(* Logix 5000 project; controller R1USB70001_CWRU_Scenario_Gen_20111116 vendor 1 type 14 code 54 rev 19.11; software revision 19.01 *)

TASK MainTask (continuous, watchdog 500 ms) : MainProgram

MODULES
   Local : vendor 1 type 14 code 54 (ICP 2, rev 19.11)
      CNB_Scenario_Generator : vendor 1 type 12 code 21 (ICP 0, rev 20.13)
         ACNR_SP_SG_N3 : vendor 1 type 12 code 111 (ControlNet 3, rev 1.83, Output RPI 8 ms)
            OB8_SP_SG_S3 : 1734-OE2V (PointIO 3, rev 3.5, Output RPI 8 ms)
            OB8_SP_SG_S2 : 1734-OB8 (PointIO 2, rev 3.22)
            OB8_SP_SG_S1 : 1734-OB8 (PointIO 1, rev 3.22)
         ACNR_RP_SG_N4 : vendor 1 type 12 code 111 (ControlNet 4, rev 1.83, Output RPI 8 ms)
            OB8_RP_SG_S1 : 1734-OB8 (PointIO 1, rev 3.22)
            OB8_RP_SG_S2 : 1734-OB8 (PointIO 2, rev 3.22)
            OB8_RP_SG_S3 : 1734-OB8 (PointIO 3, rev 3.22)
            OB8_RP_SG_S5 : 1734-OB8 (PointIO 5, rev 3.22)
            OB8_RP_SG_S6 : 1734-OB8 (PointIO 6, rev 3.22)
            OB8_RP_SG_S4 : 1734-OB8 (PointIO 4, rev 3.22)
         ACNR_GP_SG_N2 : vendor 1 type 12 code 111 (ControlNet 2, rev 1.83, Output RPI 8 ms)
            OB8_GP_SG_S1 : 1734-OB8 (PointIO 1, rev 3.22)
            OB8_GP_SG_S2 : 1734-OB8 (PointIO 2, rev 3.22)
            OB8_GP_SG_S3 : 1734-OB8 (PointIO 3, rev 3.22)
            OB8_GP_SG_S5 : 1734-OB8 (PointIO 5, rev 3.22)
            OB8_GP_SG_S4 : 1734-OB8 (PointIO 4, rev 3.22)
            OB8_GP_SG_S6 : 1734-OB8 (PointIO 6, rev 3.22)
         ACNR_CP_SG_N5 : vendor 1 type 12 code 111 (ControlNet 5, rev 1.83, Output RPI 8 ms)
            OB8_CP_SG_S1 : 1734-OB8 (PointIO 1, rev 3.22)
            OB8_CP_SG_S2 : 1734-OB8 (PointIO 2, rev 3.22)
            OB8_CP_SG_S3 : 1734-OB8 (PointIO 3, rev 3.22)
            OB8_CP_SG_S4 : 1734-OB8 (PointIO 4, rev 3.22)
            OB8_CP_SG_S5 : 1734-OB8 (PointIO 5, rev 3.22)
            OB8_CP_SG_S6 : 1734-OB8 (PointIO 6, rev 3.22)
      EN2T_Scenario_Generator : 1756-EN2T (ICP 1, Ethernet 10.88.0.101, rev 4.3)
END_MODULES

TYPE AOI_Tags :   // Tags for control of the Add-On Instructions
STRUCT
   AP_GP_SR : Cycle_Three_State;
   AP_GP_CH : Cycle_Three_State;
   WF_GP_BT : Cycle_Three_State;
   WF_GP_GD : Cycle_Three_State;
   WT_GP_BT : Cycle_Three_State;
   WT_GP_GD : Cycle_Three_State;
   SF_GP_BT : Cycle_Three_State;
   SF_GP_GD : Cycle_Three_State;
   SC_GP_BT : Cycle_Three_State;
   SC_GP_GD : Cycle_Three_State;
   RL_GP_SC : Cycle_Three_State;
   RL_GP_SF : Cycle_Three_State;
   RL_GP_WT : Cycle_Three_State;
   RL_GP_WF : Cycle_Three_State;
   CL_GP_SC : Cycle_Three_State;
   CL_GP_SF : Cycle_Three_State;
   CL_GP_WT : Cycle_Three_State;
   CL_GP_WF : Cycle_Three_State;
   IL_GP_SC : Cycle_Three_State;
   IL_GP_SF : Cycle_Three_State;
   IL_GP_WT : Cycle_Three_State;
   IL_GP_WF : Cycle_Three_State;
   AS_SP_L1 : Cycle_Three_State;
   AS_SP_L2 : Cycle_Three_State;
   WF_SP_LN : Cycle_Three_State;
   WT_SP_LN : Cycle_Three_State;
   SF_SP_LN : Cycle_Three_State;
   SC_SP_LN : Cycle_Three_State;
   RL_LP_ML_SG : Cycle_Two_State;
   RL_LP_B1_SG : Cycle_Two_State;
   RL_LP_B1_L1 : Cycle_Three_State;
   RL_LP_B1_L2 : Cycle_Three_State;
   RL_LP_B1_L3 : Cycle_Three_State;
   RL_LP_B1_L4 : Cycle_Three_State;
   RL_LP_B1_L5 : Cycle_Three_State;
   RL_LP_B2_SG : Cycle_Two_State;
   RL_LP_B2_L1 : Cycle_Three_State;
   RL_LP_B2_L2 : Cycle_Three_State;
   RL_LP_B2_L3 : Cycle_Three_State;
   RL_LP_B2_L4 : Cycle_Three_State;
   RL_LP_B2_L5 : Cycle_Three_State;
   RL_LP_B3_SG : Cycle_Two_State;
   RL_LP_B3_L1 : Cycle_Three_State;
   RL_LP_B3_L2 : Cycle_Three_State;
   RL_LP_B3_L3 : Cycle_Three_State;
   RL_LP_B3_L4 : Cycle_Three_State;
   RL_LP_B3_L5 : Cycle_Three_State;
   RL_LP_B4_SG : Cycle_Two_State;
   RL_LP_B4_L1 : Cycle_Three_State;
   RL_LP_B4_L2 : Cycle_Three_State;
   RL_LP_B4_L3 : Cycle_Three_State;
   RL_LP_B4_L4 : Cycle_Three_State;
   RL_LP_B4_L5 : Cycle_Three_State;
   CL_LP_ML_SG : Cycle_Two_State;
   CL_LP_B1_SG : Cycle_Two_State;
   CL_LP_B1_L1 : Cycle_Three_State;
   CL_LP_B1_L2 : Cycle_Three_State;
   CL_LP_B1_L3 : Cycle_Three_State;
   CL_LP_B1_L4 : Cycle_Three_State;
   CL_LP_B1_L5 : Cycle_Three_State;
   CL_LP_B2_SG : Cycle_Two_State;
   CL_LP_B2_L1 : Cycle_Three_State;
   CL_LP_B2_L2 : Cycle_Three_State;
   CL_LP_B2_L3 : Cycle_Three_State;
   CL_LP_B2_L4 : Cycle_Three_State;
   CL_LP_B2_L5 : Cycle_Three_State;
   IL_LP_ML_SG : Cycle_Two_State;
   IL_LP_B1_SG : Cycle_Two_State;
   IL_LP_B1_L1 : Cycle_Three_State;
   IL_LP_B1_L2 : Cycle_Three_State;
   IL_LP_B1_L3 : Cycle_Three_State;
   IL_LP_B1_L4 : Cycle_Three_State;
   IL_LP_B1_L5 : Cycle_Three_State;
   IL_LP_B2_SG : Cycle_Two_State;
   IL_LP_B2_L1 : Cycle_Three_State;
   IL_LP_B2_L2 : Cycle_Three_State;
   IL_LP_B2_L3 : Cycle_Three_State;
   IL_LP_B2_L4 : Cycle_Three_State;
   IL_LP_B2_L5 : Cycle_Three_State;
END_STRUCT
END_TYPE

TYPE ControlModeCmd :   // Command Bits for Control Mode
STRUCT
   Request_Scenario_Control : BOOL;   // Request for Scenario (internal) Control from the HMI
   Request_Alternate_Control : BOOL;   // Request for Alternate (external) Control from the HMI
END_STRUCT
END_TYPE

TYPE ControlModeCnx :   // Connections for Control Mode
STRUCT
   Alternate_Control_Buffer : Output_Array;   // Array of bit-defined words from Alternate (external) Control source
   Scenario_Control_Buffer : Output_Array;   // Array of bit-defined words from Scenario (internal) Control source
END_STRUCT
END_TYPE

TYPE ControlModeEv :   // Private Events for Control Mode
STRUCT
   Request_Scenario_Control : BOOL;   // Request for Scenario (internal) Control from the HMI
   Request_Alternate_Control : BOOL;   // Request for Alternate (external) Control from the HMI
   Alternate_Control_Active : BOOL;   // Alternate (external) Control is Active
END_STRUCT
END_TYPE

TYPE ControlModePub :   // Public Interface for Control Mode
STRUCT
   Cmd : ControlModeCmd;   // Command Bits for ControlMode
   Sts : ControlModeSts;   // Status bits for ControlMode
   Val : ControlModeVal;   // Values for ControlMode
END_STRUCT
END_TYPE

TYPE ControlModePv :   // Private Variables for Control Mode
STRUCT
   Cnx : ControlModeCnx;   // Connections for ControlMode
   Comments : DINT[2];   // Comment Bits
   Ev : ControlModeEv;   // Events for ControlMode
   OneShot : DINT[2];   // One Shot Bits
END_STRUCT
END_TYPE

TYPE ControlModeSts :   // Status bits for Control Mode
STRUCT
   Scenario_Control_Active : BOOL;   // Scenario (internal) Control is Active
   Alternate_Control_Active : BOOL;   // Alternate (external) Control is Active
END_STRUCT
END_TYPE

TYPE ControlModeVal :   // Values for publishing on public interface for Control Mode
STRUCT
   Active_Output_Buffer : Output_Array;   // Buffer Array of bit-defined words that are continuously mapped to real outputs
END_STRUCT
END_TYPE

TYPE DiscreteOutputsCnx :   // Connections for Discrete Outputs
STRUCT
   Active_Output_Buffer : Output_Array;   // Buffer Array of bit-defined words that are continuously mapped to real outputs
END_STRUCT
END_TYPE

TYPE DiscreteOutputsPv :   // Private Variables for Discrete Outputs
STRUCT
   Comments : DINT[2];   // Comment Bits
   Cnx : DiscreteOutputsCnx;
END_STRUCT
END_TYPE

TYPE EditScenarioCmd :   // Command Bits for EditScenario
STRUCT
   Trig_AP_GP_SR : BOOL;
   Trig_AP_GP_CH : BOOL;
   Trig_WF_GP_BT : BOOL;
   Trig_WF_GP_GD : BOOL;
   Trig_WT_GP_BT : BOOL;
   Trig_WT_GP_GD : BOOL;
   Trig_SF_GP_BT : BOOL;
   Trig_SF_GP_GD : BOOL;
   Trig_SC_GP_BT : BOOL;
   Trig_SC_GP_GD : BOOL;
   Trig_RL_GP_SC : BOOL;
   Trig_RL_GP_SF : BOOL;
   Trig_RL_GP_WT : BOOL;
   Trig_RL_GP_WF : BOOL;
   Trig_CL_GP_SC : BOOL;
   Trig_CL_GP_SF : BOOL;
   Trig_CL_GP_WT : BOOL;
   Trig_CL_GP_WF : BOOL;
   Trig_IL_GP_SC : BOOL;
   Trig_IL_GP_SF : BOOL;
   Trig_IL_GP_WT : BOOL;
   Trig_IL_GP_WF : BOOL;
   Trig_AS_SP_L1 : BOOL;
   Trig_AS_SP_L2 : BOOL;
   Trig_WF_SP_LN : BOOL;
   Trig_WT_SP_LN : BOOL;
   Trig_SF_SP_LN : BOOL;
   Trig_SC_SP_LN : BOOL;
   Trig_RL_LP_ML : BOOL;
   Trig_RL_LP_B1 : BOOL;
   Trig_RL_LP_B1_L1 : BOOL;
   Trig_RL_LP_B1_L2 : BOOL;
   Trig_RL_LP_B1_L3 : BOOL;
   Trig_RL_LP_B1_L4 : BOOL;
   Trig_RL_LP_B1_L5 : BOOL;
   Trig_RL_LP_B2 : BOOL;
   Trig_RL_LP_B2_L1 : BOOL;
   Trig_RL_LP_B2_L2 : BOOL;
   Trig_RL_LP_B2_L3 : BOOL;
   Trig_RL_LP_B2_L4 : BOOL;
   Trig_RL_LP_B2_L5 : BOOL;
   Trig_RL_LP_B3 : BOOL;
   Trig_RL_LP_B3_L1 : BOOL;
   Trig_RL_LP_B3_L2 : BOOL;
   Trig_RL_LP_B3_L3 : BOOL;
   Trig_RL_LP_B3_L4 : BOOL;
   Trig_RL_LP_B3_L5 : BOOL;
   Trig_RL_LP_B4 : BOOL;
   Trig_RL_LP_B4_L1 : BOOL;
   Trig_RL_LP_B4_L2 : BOOL;
   Trig_RL_LP_B4_L3 : BOOL;
   Trig_RL_LP_B4_L4 : BOOL;
   Trig_RL_LP_B4_L5 : BOOL;
   Trig_CL_LP_ML : BOOL;
   Trig_CL_LP_B1 : BOOL;
   Trig_CL_LP_B1_L1 : BOOL;
   Trig_CL_LP_B1_L2 : BOOL;
   Trig_CL_LP_B1_L3 : BOOL;
   Trig_CL_LP_B1_L4 : BOOL;
   Trig_CL_LP_B1_L5 : BOOL;
   Trig_CL_LP_B2 : BOOL;
   Trig_CL_LP_B2_L1 : BOOL;
   Trig_CL_LP_B2_L2 : BOOL;
   Trig_CL_LP_B2_L3 : BOOL;
   Trig_CL_LP_B2_L4 : BOOL;
   Trig_CL_LP_B2_L5 : BOOL;
   Trig_IL_LP_ML : BOOL;
   Trig_IL_LP_B1 : BOOL;
   Trig_IL_LP_B1_L1 : BOOL;
   Trig_IL_LP_B1_L2 : BOOL;
   Trig_IL_LP_B1_L3 : BOOL;
   Trig_IL_LP_B1_L4 : BOOL;
   Trig_IL_LP_B1_L5 : BOOL;
   Trig_IL_LP_B2 : BOOL;
   Trig_IL_LP_B2_L1 : BOOL;
   Trig_IL_LP_B2_L2 : BOOL;
   Trig_IL_LP_B2_L3 : BOOL;
   Trig_IL_LP_B2_L4 : BOOL;
   Trig_IL_LP_B2_L5 : BOOL;
   Next_Scenario : BOOL;
   Prev_Scenario : BOOL;
   Next_Step : BOOL;
   Prev_Step : BOOL;
   Accept_Configuration_Grid : BOOL;   // Command from the HMI to accept the current Configuration from the Grid Panel configuration screen
   Accept_Configuration_Source : BOOL;   // Command from the HMI to accept the current Configuration from the Source Panel configuration screen
   Accept_Configuration_Residential : BOOL;   // Command from the HMI to accept the current Configuration from the Residential Load Panel configuration screen
   Accept_Configuration_Commercial : BOOL;   // Command from the HMI to accept the current Configuration from the Commercial & Industrial Load Panel configuration screen
   Enter_Step_Time : BOOL;   // Enter key strobe bit from HMI for Step Time
   Enter_Scenario_Name : BOOL;   // Enter key strobe bit from HMI for Scenario Name
   Enter_Edit_Scenario_Number : BOOL;   // Enter key strobe bit from HMI for new scenario number to edit
   Enter_Edit_Step_Number : BOOL;   // Enter key strobe bit from HMI for new step number to edit
   GoToNextStep : BOOL;   // Go To Next Step in Configuration
   CopyPreviousStepGrid : BOOL;   // Command to copy the Grid configuration from the previous step
   CopyPreviousStepSource : BOOL;   // Command to copy the Source configuration from the previous step
   CopyPreviousStepResidential : BOOL;   // Command to copy the Residential configuration from the previous step
   CopyPreviousStepCommercial : BOOL;   // Command to copy the Commercial & Industrial configuration from the previous step
END_STRUCT
END_TYPE

TYPE EditScenarioDiag :   // Diagnostics for EditScenario Class
STRUCT
   StepTimeOutOfRange : BOOL;   // The requested step time is out of range. Valid range is 0 - 300 (sec).
END_STRUCT
END_TYPE

TYPE EditScenarioEv :   // Private Events for GenericObject
STRUCT
   LastStepDone : BOOL;   // Last Step Done in the Execution
   Enter_Step_Time : BOOL;   // Enter key strobe bit from HMI for Step Time
   Enter_Scenario_Name : BOOL;   // Enter key strobe bit from HMI for Scenario Name
   StepTimeOutOfRange : BOOL;   // The requested step time is out of range. Valid range is 0 - 300 (sec).
   Grid_Configuration_Accepted : BOOL;   // Grid Configuration has been accepted
   Source_Configuration_Accepted : BOOL;   // Source Configuration has been accepted
   Residential_Configuration_Accepted : BOOL;   // Residential Configuration has been accepted
   Industrial_Configuration_Accepted : BOOL;   // Industrial Configuration has been accepted
   ScenarioNumberChanged : BOOL;   // Scenario Number Changed (one scan)
   StepNumberChanged : BOOL;   // Step Number Changed (one scan)
END_STRUCT
END_TYPE

TYPE EditScenarioIntrnl :   // Internal Values for EditScenario
STRUCT
   Old_Scenario_Number : DINT;
   Old_Scenario_Step : DINT;
   Scenario_Number_Entering : DINT;
   Step_Number_Running : DINT;
   Next_Step : BOOL;
   Last_Run : BOOL;
   Scenario_Name_Entered : STRING;   // Scenario Name Entered from HMI
   Step_Number_Entering : DINT;
   Scenario_Number_Running : DINT;
   AOI_Tg : AOI_Tags;
   Scenario_Edit_Buffer : Scenario_Step;   // Edit Buffer for the Scenario Step currently being editted
   Edit_Scenario_Number : DINT;   // Scenario Number currently being editted
   Edit_Step_Number : DINT;   // Step Number currently being editted
   Step_Time_Config : DINT;   // Step Time - As Configured - No Multiplier (sec)
   Requested_Step_Time : DINT;   // Requested Step Time from HMI (sec)
   Step_Time_Diag_Timer : TIMER;   // Off-delay timer for diagnostic message for Step Time Out of Range
   Edit_Prev_Step_Number : DINT;   // Step Number previous to the one currently being editted
END_STRUCT
END_TYPE

TYPE EditScenarioPub :   // Public Interface for EditScenario
STRUCT
   Cmd : EditScenarioCmd;   // Command Bits for EditScenario
   Diag : EditScenarioDiag;   // Diagnostic bits for EditScenario
   Set : EditScenarioSet;   // Settings for EditScenario
   Sts : EditScenarioSts;   // Status bits for Edit Scenario Class
   Val : EditScenarioVal;   // Values for EditScenario
END_STRUCT
END_TYPE

TYPE EditScenarioPv :   // Private Variables for EditScenario
STRUCT
   Comments : DINT[2];   // Comment Bits
   Ev : EditScenarioEv;   // Events for EditScenario
   Intrnl : EditScenarioIntrnl;   // Internal private values for EditScenario
   OneShot : DINT[2];   // One Shot Bits
END_STRUCT
END_TYPE

TYPE EditScenarioSet :   // Settings for EditScenario class
STRUCT
   Step_Time : DINT;   // Configured Step Time Entry from HMI
   Scenario_Name_Entered : STRING;   // Scenario Name Entered from HMI
   Edit_Step_Number_Entered : DINT;   // Step Number to edit Entered from HMI
   Edit_Scenario_Number_Entered : DINT;   // Scenario Number to edit Entered from HMI
   CurrentScreenNumber : DINT;   // Current Screen Number from HMI
END_STRUCT
END_TYPE

TYPE EditScenarioSts :   // Status bits for Edit Scenario Class
STRUCT
   Grid_Configuration_Accepted : BOOL;   // Grid Configuration has been accepted
   Source_Configuration_Accepted : BOOL;   // Source Configuration has been accepted
   Residential_Configuration_Accepted : BOOL;   // Residential Configuration has been accepted
   Industrial_Configuration_Accepted : BOOL;   // Industrial Configuration has been accepted
END_STRUCT
END_TYPE

TYPE EditScenarioVal :   // Values for publishing on public interface for EditScenario
STRUCT
   Time_Multiplier : REAL;
   Scenario_Edit_Buffer : Scenario_Step;   // Edit Buffer for the Scenario Step currently being editted
   Edit_Scenario_Number : DINT;   // Scenario Number currently being editted
   Edit_Step_Number : DINT;   // Step Number currently being editted
   Edit_Scenario_Name : STRING;   // Name of Scenario currently being editted
END_STRUCT
END_TYPE

TYPE ExecuteCmd :   // Command Bits for Execute
STRUCT
   Run : BOOL;   // Run Command from HMI
   Stop : BOOL;   // Stop Command from HMI
   Skip : BOOL;   // Skip Command from HMI
   Resume : BOOL;   // Resume Command from HMI
   Pause : BOOL;   // Pause Command from HMI
   Enter_Scenario_Start_Number : BOOL;   // Enter key strobe bit from HMI for Scenario Start Number
   Enter_Scenario_Stop_Number : BOOL;   // Enter key strobe bit from HMI for Scenario Stop Number
   Enter_Step_Start_Number : BOOL;   // Enter key strobe bit from HMI for Step Start Number
   Enter_Step_Stop_Number : BOOL;   // Enter key strobe bit from HMI for Step Stop Number
   Enter_Time_Multiplier : BOOL;   // Enter key strobe bit from HMI for Scenario Time Multiplier
END_STRUCT
END_TYPE

TYPE ExecuteDiag :   // Diagnostics for Execute Class
STRUCT
   TimeMultiplierOutOfRange : BOOL;   // The requested time multiplier is out of range. Valid range is 1 - 100 (0.1 sec).
   StartAfterStop : BOOL;   // The requested Start Scenario or Start Step is after the current Stop Scenario and Stop Step.
   StopBeforeStart : BOOL;   // The requested Stop Scenario or Stop Step is before the current Start Scenario and Start Step.
   StartScenarioOutOfRange : BOOL;   // The requested Start Scenario number is out of range (1 - 99)
   StartStepOutOfRange : BOOL;   // The requested Start Step number is out of range (1 - 99)
   StopScenarioOutOfRange : BOOL;   // The requested Stop Scenario number is out of range (1 - 99)
   StopStepOutOfRange : BOOL;   // The requested Stop Step number is out of range (1 - 99)
END_STRUCT
END_TYPE

TYPE ExecuteEv :   // Private Events for Execute
STRUCT
   Tr : BOOL;   // State Transition Bit
   LastStepDone : BOOL;   // Last Step Done in the Execution
   Run : BOOL;   // Run Command from HMI - Ev 1
   Stop : BOOL;   // Stop Command from HMI - Ev 4
   Skip : BOOL;   // Skip Command from HMI
   Resume : BOOL;   // Resume Command from HMI - Ev 3
   Pause : BOOL;   // Pause Command from HMI - Ev 2
   Enter_Scenario_Start_Number : BOOL;   // Enter key strobe bit from HMI for Scenario Start Number
   Enter_Scenario_Stop_Number : BOOL;   // Enter key strobe bit from HMI for Scenario Stop Number
   Enter_Step_Start_Number : BOOL;   // Enter key strobe bit from HMI for Step Start Number
   Enter_Step_Stop_Number : BOOL;   // Enter key strobe bit from HMI for Step Stop Number
   Enter_Time_Multiplier : BOOL;   // Enter key strobe bit from HMI for Scenario Time Multiplier
   TimeMultiplierOutOfRange : BOOL;   // The requested time multiplier is out of range. Valid range is 1 - 100 (0.1 sec).
   StartAfterStop : BOOL;   // The requested Start Scenario or Start Step is after the current Stop Scenario and Stop Step.
   StopBeforeStart : BOOL;   // The requested Stop Scenario or Stop Step is before the current Start Scenario and Start Step.
   StartScenarioOutOfRange : BOOL;   // The requested Start Scenario number is out of range (1 - 99)
   StartStepOutOfRange : BOOL;   // The requested Start Step number is out of range (1 - 99)
   StopScenarioOutOfRange : BOOL;   // The requested Stop Scenario number is out of range (1 - 99)
   StopStepOutOfRange : BOOL;   // The requested Stop Step number is out of range (1 - 99)
END_STRUCT
END_TYPE

TYPE ExecuteIntrnl :   // Internal Values for Execute
STRUCT
   Current_Step_Number : DINT;   // Step number currently executing or selected to execute
   Current_Scenario_Number : DINT;   // Scenario number currently executing or selected to execute
   Scenario_Start_Number : DINT;   // Scenario Start Number
   Scenario_Stop_Number : DINT;   // Scenario Stop Number
   Step_Start_Number : DINT;   // Step Start Number
   Step_Stop_Number : DINT;   // Step Stop Number
   Time_Multiplier : DINT;   // Time Multiplier for scenario execution. Scaled. (0.1 sec)
   Step_Timer : TIMER;   // Step Timer for currently executing step
   Scenario_Control_Buffer : Output_Array;   // Output buffer from Scenario Execution
   Actual_Step_Time : DINT;
   Configured_Scenario_Time : DINT;
   Actual_Scenario_Time : DINT;
   Total_Scenario_Time_Config : DINT;   // Total Scenario Time - As Configured - No Multiplier (sec)
   Scenario_Time_Remaining_Config : DINT;   // Scenario Time Remaining - As Configured - No Multiplier (sec)
   Total_Step_Time_Config : DINT;   // Total Step Time - As Configured - No Multiplier (sec)
   Step_Time_Remaining_Config : DINT;   // Step Time Remaining - As Configured - No Multiplier (sec)
   Total_Scenario_Time_Actual : DINT;   // Total Scenario Time - Actual - Includes Multiplier (0.1 sec)
   Scenario_Time_Remaining_Actual : DINT;   // Scenario Time Remaining - Actual - Includes Multiplier (0.1 sec)
   Total_Step_Time_Actual : DINT;   // Total Step Time - Actual - Includes Multiplier (0.1 sec)
   Step_Time_Remaining_Actual : DINT;   // Step Time Remaining - Actual - Includes Multiplier (0.1 sec)
   Virtual_Start_Step : DINT;   // Start Scenario * 100 + Start Step = Virtual Start Step
   Virtual_Stop_Step : DINT;   // Stop Scenario * 100 + Stop Step = Virtual Stop Step
   Virtual_Current_Step : DINT;   // Current Scenario * 100 + Current Step = Virtual Current Step
   Virtual_Current_Step_Plus_1 : DINT;   // Virtual Current Step Plus 1
   Requested_Scenario_Start_Number : DINT;   // Requested Scenario Start Number (not error checked)
   Requested_Scenario_Stop_Number : DINT;   // Requested Scenario Stop Number (not error checked)
   Requested_Step_Start_Number : DINT;   // Requested Step Start Number (not error checked)
   Requested_Step_Stop_Number : DINT;   // Requested Step Stop Number (not error checked)
   Requested_Time_Multiplier : DINT;   // Requested Time Multiplier for scenario execution. Scaled. (0.1 sec) (not error checked)
   Requested_Virtual_Start_Step : DINT;   // Requested Start Scenario * 100 + Requested Start Step = Requested Virtual Start Step
   Requested_Virtual_Stop_Step : DINT;   // Requested Stop Scenario * 100 + Requested Stop Step = Requested Virtual Stop Step
   TM_Diag_Timer : TIMER;   // Off-delay timer for diagnostic message for Time Multiplier Out of Range
   SAS_Diag_Timer : TIMER;   // Off-delay timer for diagnostic message for Start Scenario or Step After Stop
   SBS_Diag_Timer : TIMER;   // Off-delay timer for diagnostic message for Stop Scenario or Step Before Start
   Start_Scenario_Diag_Timer : TIMER;   // Off-delay timer for diagnostic message for Start Scenario Out of Range
   Stop_Scenario_Diag_Timer : TIMER;   // Off-delay timer for diagnostic message for Stop Scenario Out of Range
   Start_Step_Diag_Timer : TIMER;   // Off-delay timer for diagnostic message for Start Step Out of Range
   Stop_Step_Diag_Timer : TIMER;   // Off-delay timer for diagnostic message for Stop Step Out of Range
   VirtualStepTime : DINT[10000];
   BuildTableScanCounter : DINT;
END_STRUCT
END_TYPE

TYPE ExecutePub :   // Public Interface for Execute
STRUCT
   Cmd : ExecuteCmd;   // Command Bits for Execute
   Diag : ExecuteDiag;   // Diagnostics for Execute
   Set : ExecuteSet;   // Settings for Execute
   Sts : ExecuteSts;   // Status bits for Execute
   Val : ExecuteVal;   // Values for Execute
END_STRUCT
END_TYPE

TYPE ExecutePv :   // Private Variables for Execute
STRUCT
   Comments : DINT[2];   // Comment Bits
   Ev : ExecuteEv;   // Events for Execute
   Intrnl : ExecuteIntrnl;   // Internal private values for Execute
   OneShot : DINT[2];   // One Shot Bits
   St : DINT;   // States for Execute
END_STRUCT
END_TYPE

TYPE ExecuteSet :   // Settings for Execute Class
STRUCT
   Scenario_Start_Number : DINT;   // Scenario Start Number
   Scenario_Stop_Number : DINT;   // Scenario Stop Number
   Step_Start_Number : DINT;   // Step Start Number
   Step_Stop_Number : DINT;   // Step Stop Number
   Time_Multiplier : DINT;   // Time Multiplier for scenario execution. Scaled. (0.1 sec)
END_STRUCT
END_TYPE

TYPE ExecuteSts :   // Status bits for Execute
STRUCT
   Running : BOOL;   // Scenario Execution is Running
   Paused : BOOL;   // Scenario Execution is Paused (timer paused, but outputs active)
   Stopped : BOOL;   // Scenario Execution is Stopped (all outputs off)
END_STRUCT
END_TYPE

TYPE ExecuteVal :   // Values for publishing on public interface for Execute
STRUCT
   Scenario_Control_Buffer : Output_Array;   // Output buffer from Scenario Execution
   Total_Scenario_Time_Config : DINT;   // Total Scenario Time - As Configured - No Multiplier (sec)
   Scenario_Time_Remaining_Config : DINT;   // Scenario Time Remaining - As Configured - No Multiplier (sec)
   Total_Step_Time_Config : DINT;   // Total Step Time - As Configured - No Multiplier (sec)
   Step_Time_Remaining_Config : DINT;   // Step Time Remaining - As Configured - No Multiplier (sec)
   Total_Scenario_Time_Actual : DINT;   // Total Scenario Time - Actual - Includes Multiplier (0.1 sec)
   Scenario_Time_Remaining_Actual : DINT;   // Scenario Time Remaining - Actual - Includes Multiplier (0.1 sec)
   Total_Step_Time_Actual : DINT;   // Total Step Time - Actual - Includes Multiplier (0.1 sec)
   Step_Time_Remaining_Actual : DINT;   // Step Time Remaining - Actual - Includes Multiplier (0.1 sec)
   Time_Multiplier : DINT;   // Time Multiplier for scenario execution. Scaled. (0.1 sec)
   Current_Step_Number : DINT;   // Step number currently executing or selected to execute
   Current_Scenario_Number : DINT;   // Scenario number currently executing or selected to execute
   Scenario_Start_Number : DINT;   // Scenario Start Number
   Scenario_Stop_Number : DINT;   // Scenario Stop Number
   Step_Start_Number : DINT;   // Step Start Number
   Step_Stop_Number : DINT;   // Step Stop Number
   Scenario_Name_Running : STRING;   // Name of Scenario currently running or scheduled to run
END_STRUCT
END_TYPE

TYPE HMICnx :   // Connections for HMI
STRUCT
   Active_Output_Buffer : Output_Array;   // Buffer Array of bit-defined words that are continuously mapped to real outputs
END_STRUCT
END_TYPE

TYPE HMIIntrnl :   // Internal values for HMI Class
STRUCT
   RequestedScreenNumber : DINT;   // Screen Number Requested by another softwsare class
   ScreenNumberRequestToHMI : DINT;   // Screen Number Request sent to HMI
END_STRUCT
END_TYPE

TYPE HMIPub :   // Public Interface for HMI
STRUCT
   Set : HMISet;   // Settings for HMIPub
   Val : HMIVal;   // Values for HMIPub
END_STRUCT
END_TYPE

TYPE HMIPv :   // Private Variables for HMI
STRUCT
   Cnx : HMICnx;   // Connections for HMIPv
   Comments : DINT[2];   // Comment Bits
   Ev : EditScenarioEv;   // Events for HMIPv
   Intrnl : HMIIntrnl;   // Internal values for HMI Class
   OneShot : DINT[2];   // One Shot Bits
END_STRUCT
END_TYPE

TYPE HMISet :   // Settings for HMI
STRUCT
   HMI_Intfc_WRITE_Buffer : DINT[20];   // Write Buffer for HMI to Write to as a contiguous block of memory (array of DINTs)
   HMI_Intfc_String_WRITE_Buffer : STRING;   // Write Buffer for HMI to Write to as a contiguous block of memory (single STRING tag)
END_STRUCT
END_TYPE

TYPE HMIVal :   // Values for publishing on public interface for HMI
STRUCT
   HMI_Intfc_READ_Buffer : DINT[40];
   HMI_Intfc_String_READ_Buffer : STRING[2];
   CurrentScreenNumber : DINT;   // Current Screen Number reported back from HMI
END_STRUCT
END_TYPE

TYPE Output_Array :
STRUCT
   Data : DINT[8];
END_STRUCT
END_TYPE

TYPE Scenario_Def :   // Define a Single Scenario
STRUCT
   Name : STRING;
   Step : Scenario_Step[100];
END_STRUCT
END_TYPE

TYPE Scenario_Step :   // Define a step in a scenario
STRUCT
   Output_Table : Output_Array;
   Configured_Step_Time : DINT;
END_STRUCT
END_TYPE

ADD_ON_INSTRUCTION Cycle_Three_State   (* revision 1.0 *)
// Cycles the two Scenario bits relating to a Normally Open and Normally Closed relay pair from the Scenario Generator through three valid states.
VAR_IN_OUT
   Trigger : BOOL; {required}   // Command from the HMI to advance to the next state in order
   NO : BOOL; {required}   // Output for the Normally Open (bypass) Relay of the NO/NC pair of scenario generator relays
   NC : BOOL; {required}   // Output for the Normally Closed (blocking) Relay of the NO/NC pair of scenario generator relays
END_VAR
VAR
   State : DINT;   // State of NC/NO pair of relays from Scenario Generator
        .0   // State of NO relay from Scenario Generator
        .1   // State of NC relay from Scenario Generator
   Comment : DINT; {access None}   // Comment bit
   AdvanceOneShot : BOOL; {access None}   // One Shot instruction to advance only one state per button press
END_VAR

ROUTINE Logic   (* ladder *)
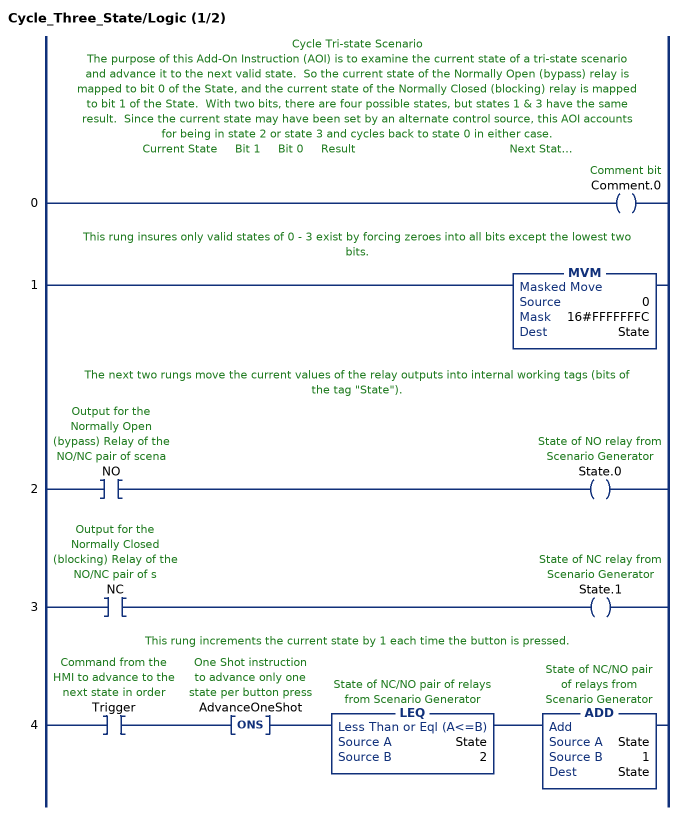
   // Cycle Tri-state Scenario
   // The purpose of this Add-On Instruction (AOI) is to examine the current state of a tri-state scenario and advance it to the next valid state.  So the current state of the Normally Open (bypass) relay is mapped to bit 0 of the State, and the current state of the Normally Closed (blocking) relay is mapped to bit 1 of the State.  With two bits, there are four possible states, but states 1 & 3 have the same result.  Since the current state may have been set by an alternate control source, this AOI accounts for being in state 2 or state 3 and cycles back to state 0 in either case.
   // Current State     Bit 1     Bit 0     Result                                            Next State
   //     0                 0          0       Student Control                                      1
   //     1                 0          1      Bypassed (Forced On)                          2
   //     2                 1          0       Blocked (Forced Off)                            0
   //     3                 1          1       Bypassed (Forced On)                         0
   0: OTE(Comment.0);
   // This rung insures only valid states of 0 - 3 exist by forcing zeroes into all bits except the lowest two bits.
   1: MVM(0,16#FFFFFFFC,State);
   // The next two rungs move the current values of the relay outputs into internal working tags (bits of the tag "State").
   2: XIC(NO)OTE(State.0);
   3: XIC(NC)OTE(State.1);
   // This rung increments the current state by 1 each time the button is pressed.
   4: XIC(Trigger)ONS(AdvanceOneShot)LEQ(State,2)ADD(State,1,State);
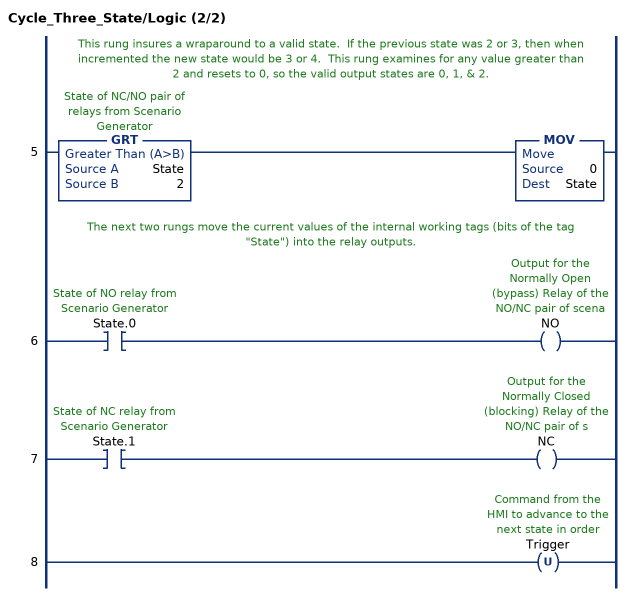
   // This rung insures a wraparound to a valid state.  If the previous state was 2 or 3, then when incremented the new state would be 3 or 4.  This rung examines for any value greater than 2 and resets to 0, so the valid output states are 0, 1, & 2.
   5: GRT(State,2)MOV(0,State);
   // The next two rungs move the current values of the internal working tags (bits of the tag "State") into the relay outputs.
   6: XIC(State.0)OTE(NO);
   7: XIC(State.1)OTE(NC);
   8: OTU(Trigger);
END_ROUTINE
END_ADD_ON_INSTRUCTION

ADD_ON_INSTRUCTION Cycle_Two_State   (* revision 1.0 *)
// Cycles the output bit between the two states of on and off for a Normally Open relay.
VAR_IN_OUT
   Trigger : BOOL; {required}   // Command from the HMI to advance to the next state in order
   NO : BOOL; {required}   // Output for the Normally Open Relay from thescenario generator
END_VAR
VAR
   Temp : BOOL;   // Temporary storage bit for current state when command is triggered.
   AdvanceOneShot : BOOL; {access None}   // One Shot instruction to advance only one state per button press
   Comment : DINT; {access None}   // Comment bit
END_VAR

ROUTINE Logic   (* ladder *)
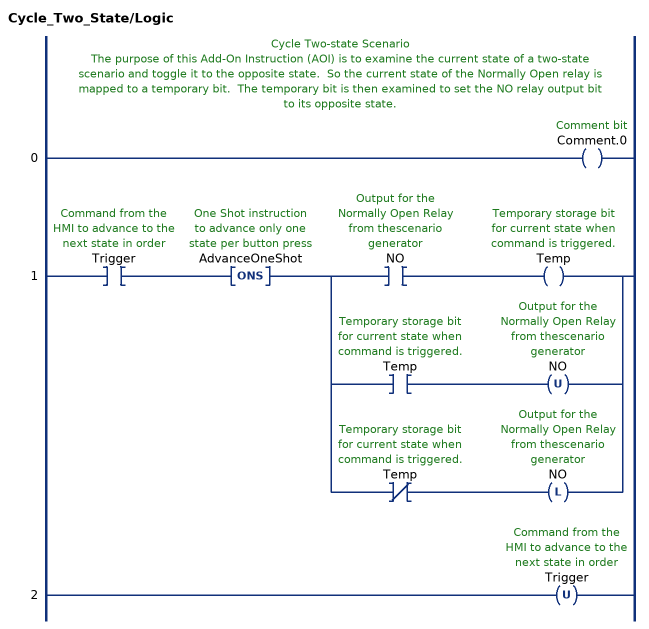
   // Cycle Two-state Scenario
   // The purpose of this Add-On Instruction (AOI) is to examine the current state of a two-state scenario and toggle it to the opposite state.  So the current state of the Normally Open relay is mapped to a temporary bit.  The temporary bit is then examined to set the NO relay output bit to its opposite state.
   0: OTE(Comment.0);
   1: XIC(Trigger)ONS(AdvanceOneShot)[XIC(NO) OTE(Temp) ,XIC(Temp) OTU(NO) ,XIO(Temp) OTL(NO) ];
   2: OTU(Trigger);
END_ROUTINE
END_ADD_ON_INSTRUCTION

VAR_GLOBAL   (* controller tags *)
   Alternate_Control_Buffer : Output_Array := (Data[1] := 1024);   // Array of bit-defined words from Alternate (external) Control source
   AP_GP_CH_SG1 : ALIAS FOR ACNR_GP_SG_N2:1:O.2;
   AP_GP_CH_SG2 : ALIAS FOR ACNR_GP_SG_N2:1:O.3;
   AP_GP_SR_SG1 : ALIAS FOR ACNR_GP_SG_N2:1:O.0;
   AP_GP_SR_SG2 : ALIAS FOR ACNR_GP_SG_N2:1:O.1;
   AS_SP_L1_SG1 : ALIAS FOR ACNR_SP_SG_N3:1:O.0;
   AS_SP_L1_SG2 : ALIAS FOR ACNR_SP_SG_N3:1:O.1;
   AS_SP_L2_SG1 : ALIAS FOR ACNR_SP_SG_N3:1:O.2;
   AS_SP_L2_SG2 : ALIAS FOR ACNR_SP_SG_N3:1:O.3;
   BuildTableIndex : DINT := 2699;
   CalcRemainTimeIndex : DINT := 281;
   CalcTotalTimeIndex : DINT := 281;
   CL_GP_SC_SG1 : ALIAS FOR ACNR_GP_SG_N2:5:O.0;
   CL_GP_SC_SG2 : ALIAS FOR ACNR_GP_SG_N2:5:O.1;
   CL_GP_SF_SG1 : ALIAS FOR ACNR_GP_SG_N2:5:O.2;
   CL_GP_SF_SG2 : ALIAS FOR ACNR_GP_SG_N2:5:O.3;
   CL_GP_WF_SG1 : ALIAS FOR ACNR_GP_SG_N2:5:O.6;
   CL_GP_WF_SG2 : ALIAS FOR ACNR_GP_SG_N2:5:O.7;
   CL_GP_WT_SG1 : ALIAS FOR ACNR_GP_SG_N2:5:O.4;
   CL_GP_WT_SG2 : ALIAS FOR ACNR_GP_SG_N2:5:O.5;
   CL_LP_B1_L1_SG1 : ALIAS FOR ACNR_CP_SG_N5:1:O.2;
   CL_LP_B1_L1_SG2 : ALIAS FOR ACNR_CP_SG_N5:1:O.3;
   CL_LP_B1_L2_SG1 : ALIAS FOR ACNR_CP_SG_N5:1:O.4;
   CL_LP_B1_L2_SG2 : ALIAS FOR ACNR_CP_SG_N5:1:O.5;
   CL_LP_B1_L3_SG1 : ALIAS FOR ACNR_CP_SG_N5:1:O.6;
   CL_LP_B1_L3_SG2 : ALIAS FOR ACNR_CP_SG_N5:1:O.7;
   CL_LP_B1_L4_SG1 : ALIAS FOR ACNR_CP_SG_N5:2:O.0;
   CL_LP_B1_L4_SG2 : ALIAS FOR ACNR_CP_SG_N5:2:O.1;
   CL_LP_B1_L5_SG1 : ALIAS FOR ACNR_CP_SG_N5:2:O.2;
   CL_LP_B1_L5_SG2 : ALIAS FOR ACNR_CP_SG_N5:2:O.3;
   CL_LP_B1_SG : ALIAS FOR ACNR_CP_SG_N5:1:O.1;
   CL_LP_B2_L1_SG1 : ALIAS FOR ACNR_CP_SG_N5:2:O.5;
   CL_LP_B2_L1_SG2 : ALIAS FOR ACNR_CP_SG_N5:2:O.6;
   CL_LP_B2_L2_SG1 : ALIAS FOR ACNR_CP_SG_N5:3:O.0;
   CL_LP_B2_L2_SG2 : ALIAS FOR ACNR_CP_SG_N5:3:O.1;
   CL_LP_B2_L3_SG1 : ALIAS FOR ACNR_CP_SG_N5:3:O.2;
   CL_LP_B2_L3_SG2 : ALIAS FOR ACNR_CP_SG_N5:3:O.3;
   CL_LP_B2_L4_SG1 : ALIAS FOR ACNR_CP_SG_N5:3:O.4;
   CL_LP_B2_L4_SG2 : ALIAS FOR ACNR_CP_SG_N5:3:O.5;
   CL_LP_B2_L5_SG1 : ALIAS FOR ACNR_CP_SG_N5:3:O.6;
   CL_LP_B2_L5_SG2 : ALIAS FOR ACNR_CP_SG_N5:3:O.7;
   CL_LP_B2_SG : ALIAS FOR ACNR_CP_SG_N5:2:O.4;
   CL_LP_ML_SG : ALIAS FOR ACNR_CP_SG_N5:1:O.0;
   ControlMode : ControlModePub := (Sts.Scenario_Control_Active := 1);
   Current_Screen_Number : INT := 3;
   EditScenario : EditScenarioPub := (Set.Step_Time := 5, Set.Scenario_Name_Entered := 'Load panels, load relays only.', Set.Edit_Step_Number_Entered := 3, Set.Edit_Scenario_Number_Entered := 3, Set.CurrentScreenNumber := 1, Val.Scenario_Edit_Buffer.Output_Table.Data[4] := 4096, Val.Scenario_Edit_Buffer.Configured_Step_Time := 5, Val.Edit_Scenario_Number := 3, Val.Edit_Step_Number := 3, Val.Edit_Scenario_Name := 'Load panels, ground fault relays only.');
   Execute : ExecutePub := (Set.Scenario_Start_Number := 1, Set.Scenario_Stop_Number := 2, Set.Step_Start_Number := 1, Set.Step_Stop_Number := 80, Set.Time_Multiplier := 10, Sts.Stopped := 1, Val.Total_Scenario_Time_Config := 740, Val.Scenario_Time_Remaining_Config := 735, Val.Total_Step_Time_Config := 5, Val.Total_Scenario_Time_Actual := 7400, Val.Scenario_Time_Remaining_Actual := 7350, Val.Total_Step_Time_Actual := 50, Val.Time_Multiplier := 10, Val.Current_Step_Number := 1, Val.Current_Scenario_Number := 1, Val.Scenario_Start_Number := 1, Val.Scenario_Stop_Number := 2, Val.Step_Start_Number := 1, Val.Step_Stop_Number := 80, Val.Scenario_Name_Running := 'Source and Grid panels, all relays.');
   HMI : HMIPub := (Set.HMI_Intfc_WRITE_Buffer[0] := 3, Set.HMI_Intfc_WRITE_Buffer[1] := 3, Set.HMI_Intfc_WRITE_Buffer[2] := 5, Set.HMI_Intfc_WRITE_Buffer[7] := 1, Set.HMI_Intfc_WRITE_Buffer[8] := 1, Set.HMI_Intfc_WRITE_Buffer[9] := 2, Set.HMI_Intfc_WRITE_Buffer[10] := 80, Set.HMI_Intfc_WRITE_Buffer[11] := 10, Set.HMI_Intfc_WRITE_Buffer[12] := 1, Set.HMI_Intfc_String_WRITE_Buffer := 'Load panels, load relays only.', Val.HMI_Intfc_READ_Buffer[0] := 1, Val.HMI_Intfc_READ_Buffer[1] := 1, Val.HMI_Intfc_READ_Buffer[2] := 3, Val.HMI_Intfc_READ_Buffer[3] := 3, Val.HMI_Intfc_READ_Buffer[4] := 5, Val.HMI_Intfc_READ_Buffer[5] := 10, Val.HMI_Intfc_READ_Buffer[6] := 740, Val.HMI_Intfc_READ_Buffer[7] := 735, Val.HMI_Intfc_READ_Buffer[8] := 5, Val.HMI_Intfc_READ_Buffer[10] := 7400, Val.HMI_Intfc_READ_Buffer[11] := 7350, Val.HMI_Intfc_READ_Buffer[12] := 50, Val.HMI_Intfc_READ_Buffer[14] := 12, Val.HMI_Intfc_READ_Buffer[16] := 2048, Val.HMI_Intfc_READ_Buffer[30] := 1, Val.HMI_Intfc_READ_Buffer[31] := 1, Val.HMI_Intfc_READ_Buffer[32] := 1, Val.HMI_Intfc_READ_Buffer[33] := 1, Val.HMI_Intfc_READ_Buffer[34] := 2, Val.HMI_Intfc_READ_Buffer[35] := 80, Val.HMI_Intfc_String_READ_Buffer[0] := 'Load panels, ground fault relays only.', Val.HMI_Intfc_String_READ_Buffer[1] := 'Source and Grid panels, all relays.', Val.CurrentScreenNumber := 1);
   HMI_Intfc_Read_Buffer : DINT[40] := ([0] := 1, [1] := 1, [2] := 3, [3] := 3, [4] := 5, [5] := 10, [6] := 740, [7] := 735, [8] := 5, [10] := 7400, [11] := 7350, [12] := 50, [14] := 12, [16] := 2048, [30] := 1, [31] := 1, [32] := 1, [33] := 1, [34] := 2, [35] := 80);
   HMI_Intfc_String_Read_Buffer : STRING[2] := ([0] := 'Load panels, ground fault relays only.', [1] := 'Source and Grid panels, all relays.');
   HMI_Intfc_String_Write_Buffer : STRING := 'Load panels, load relays only.';
   HMI_Intfc_Write_Buffer : DINT[20] := ([0] := 3, [1] := 3, [2] := 5, [7] := 1, [8] := 1, [9] := 2, [10] := 80, [11] := 10, [12] := 1);
   IL_GP_SC_SG1 : ALIAS FOR ACNR_GP_SG_N2:6:O.0;
   IL_GP_SC_SG2 : ALIAS FOR ACNR_GP_SG_N2:6:O.1;
   IL_GP_SF_SG1 : ALIAS FOR ACNR_GP_SG_N2:6:O.2;
   IL_GP_SF_SG2 : ALIAS FOR ACNR_GP_SG_N2:6:O.3;
   IL_GP_WF_SG1 : ALIAS FOR ACNR_GP_SG_N2:6:O.6;
   IL_GP_WF_SG2 : ALIAS FOR ACNR_GP_SG_N2:6:O.7;
   IL_GP_WT_SG1 : ALIAS FOR ACNR_GP_SG_N2:6:O.4;
   IL_GP_WT_SG2 : ALIAS FOR ACNR_GP_SG_N2:6:O.5;
   IL_LP_B1_L1_SG1 : ALIAS FOR ACNR_CP_SG_N5:4:O.2;
   IL_LP_B1_L1_SG2 : ALIAS FOR ACNR_CP_SG_N5:4:O.3;
   IL_LP_B1_L2_SG1 : ALIAS FOR ACNR_CP_SG_N5:4:O.4;
   IL_LP_B1_L2_SG2 : ALIAS FOR ACNR_CP_SG_N5:4:O.5;
   IL_LP_B1_L3_SG1 : ALIAS FOR ACNR_CP_SG_N5:4:O.6;
   IL_LP_B1_L3_SG2 : ALIAS FOR ACNR_CP_SG_N5:4:O.7;
   IL_LP_B1_L4_SG1 : ALIAS FOR ACNR_CP_SG_N5:5:O.0;
   IL_LP_B1_L4_SG2 : ALIAS FOR ACNR_CP_SG_N5:5:O.1;
   IL_LP_B1_L5_SG1 : ALIAS FOR ACNR_CP_SG_N5:5:O.2;
   IL_LP_B1_L5_SG2 : ALIAS FOR ACNR_CP_SG_N5:5:O.3;
   IL_LP_B1_SG : ALIAS FOR ACNR_CP_SG_N5:4:O.1;
   IL_LP_B2_L1_SG1 : ALIAS FOR ACNR_CP_SG_N5:5:O.5;
   IL_LP_B2_L1_SG2 : ALIAS FOR ACNR_CP_SG_N5:5:O.6;
   IL_LP_B2_L2_SG1 : ALIAS FOR ACNR_CP_SG_N5:6:O.0;
   IL_LP_B2_L2_SG2 : ALIAS FOR ACNR_CP_SG_N5:6:O.1;
   IL_LP_B2_L3_SG1 : ALIAS FOR ACNR_CP_SG_N5:6:O.2;
   IL_LP_B2_L3_SG2 : ALIAS FOR ACNR_CP_SG_N5:6:O.3;
   IL_LP_B2_L4_SG1 : ALIAS FOR ACNR_CP_SG_N5:6:O.4;
   IL_LP_B2_L4_SG2 : ALIAS FOR ACNR_CP_SG_N5:6:O.5;
   IL_LP_B2_L5_SG1 : ALIAS FOR ACNR_CP_SG_N5:6:O.6;
   IL_LP_B2_L5_SG2 : ALIAS FOR ACNR_CP_SG_N5:6:O.7;
   IL_LP_B2_SG : ALIAS FOR ACNR_CP_SG_N5:5:O.4;
   IL_LP_ML_SG : ALIAS FOR ACNR_CP_SG_N5:4:O.0;
   Request_Screen_Number : INT;
   RL_GP_SC_SG1 : ALIAS FOR ACNR_GP_SG_N2:4:O.0;
   RL_GP_SC_SG2 : ALIAS FOR ACNR_GP_SG_N2:4:O.1;
   RL_GP_SF_SG1 : ALIAS FOR ACNR_GP_SG_N2:4:O.2;
   RL_GP_SF_SG2 : ALIAS FOR ACNR_GP_SG_N2:4:O.3;
   RL_GP_WF_SG1 : ALIAS FOR ACNR_GP_SG_N2:4:O.6;
   RL_GP_WF_SG2 : ALIAS FOR ACNR_GP_SG_N2:4:O.7;
   RL_GP_WT_SG1 : ALIAS FOR ACNR_GP_SG_N2:4:O.4;
   RL_GP_WT_SG2 : ALIAS FOR ACNR_GP_SG_N2:4:O.5;
   RL_LP_B1_L1_SG1 : ALIAS FOR ACNR_RP_SG_N4:1:O.2;
   RL_LP_B1_L1_SG2 : ALIAS FOR ACNR_RP_SG_N4:1:O.3;
   RL_LP_B1_L2_SG1 : ALIAS FOR ACNR_RP_SG_N4:1:O.4;
   RL_LP_B1_L2_SG2 : ALIAS FOR ACNR_RP_SG_N4:1:O.5;
   RL_LP_B1_L3_SG1 : ALIAS FOR ACNR_RP_SG_N4:1:O.6;
   RL_LP_B1_L3_SG2 : ALIAS FOR ACNR_RP_SG_N4:1:O.7;
   RL_LP_B1_L4_SG1 : ALIAS FOR ACNR_RP_SG_N4:2:O.0;
   RL_LP_B1_L4_SG2 : ALIAS FOR ACNR_RP_SG_N4:2:O.1;
   RL_LP_B1_L5_SG1 : ALIAS FOR ACNR_RP_SG_N4:2:O.2;
   RL_LP_B1_L5_SG2 : ALIAS FOR ACNR_RP_SG_N4:2:O.3;
   RL_LP_B1_SG : ALIAS FOR ACNR_RP_SG_N4:1:O.1;
   RL_LP_B2_L1_SG1 : ALIAS FOR ACNR_RP_SG_N4:2:O.5;
   RL_LP_B2_L1_SG2 : ALIAS FOR ACNR_RP_SG_N4:2:O.6;
   RL_LP_B2_L2_SG1 : ALIAS FOR ACNR_RP_SG_N4:2:O.7;
   RL_LP_B2_L2_SG2 : ALIAS FOR ACNR_RP_SG_N4:3:O.0;
   RL_LP_B2_L3_SG1 : ALIAS FOR ACNR_RP_SG_N4:3:O.1;
   RL_LP_B2_L3_SG2 : ALIAS FOR ACNR_RP_SG_N4:3:O.2;
   RL_LP_B2_L4_SG1 : ALIAS FOR ACNR_RP_SG_N4:3:O.3;
   RL_LP_B2_L4_SG2 : ALIAS FOR ACNR_RP_SG_N4:3:O.4;
   RL_LP_B2_L5_SG1 : ALIAS FOR ACNR_RP_SG_N4:3:O.5;
   RL_LP_B2_L5_SG2 : ALIAS FOR ACNR_RP_SG_N4:3:O.6;
   RL_LP_B2_SG : ALIAS FOR ACNR_RP_SG_N4:2:O.4;
   RL_LP_B3_L1_SG1 : ALIAS FOR ACNR_RP_SG_N4:4:O.0;
   RL_LP_B3_L1_SG2 : ALIAS FOR ACNR_RP_SG_N4:4:O.1;
   RL_LP_B3_L2_SG1 : ALIAS FOR ACNR_RP_SG_N4:4:O.2;
   RL_LP_B3_L2_SG2 : ALIAS FOR ACNR_RP_SG_N4:4:O.3;
   RL_LP_B3_L3_SG1 : ALIAS FOR ACNR_RP_SG_N4:4:O.4;
   RL_LP_B3_L3_SG2 : ALIAS FOR ACNR_RP_SG_N4:4:O.5;
   RL_LP_B3_L4_SG1 : ALIAS FOR ACNR_RP_SG_N4:4:O.6;
   RL_LP_B3_L4_SG2 : ALIAS FOR ACNR_RP_SG_N4:4:O.7;
   RL_LP_B3_L5_SG1 : ALIAS FOR ACNR_RP_SG_N4:5:O.0;
   RL_LP_B3_L5_SG2 : ALIAS FOR ACNR_RP_SG_N4:5:O.1;
   RL_LP_B3_SG : ALIAS FOR ACNR_RP_SG_N4:3:O.7;
   RL_LP_B4_L1_SG1 : ALIAS FOR ACNR_RP_SG_N4:5:O.3;
   RL_LP_B4_L1_SG2 : ALIAS FOR ACNR_RP_SG_N4:5:O.4;
   RL_LP_B4_L2_SG1 : ALIAS FOR ACNR_RP_SG_N4:5:O.5;
   RL_LP_B4_L2_SG2 : ALIAS FOR ACNR_RP_SG_N4:5:O.6;
   RL_LP_B4_L3_SG1 : ALIAS FOR ACNR_RP_SG_N4:5:O.7;
   RL_LP_B4_L3_SG2 : ALIAS FOR ACNR_RP_SG_N4:6:O.0;
   RL_LP_B4_L4_SG1 : ALIAS FOR ACNR_RP_SG_N4:6:O.1;
   RL_LP_B4_L4_SG2 : ALIAS FOR ACNR_RP_SG_N4:6:O.2;
   RL_LP_B4_L5_SG1 : ALIAS FOR ACNR_RP_SG_N4:6:O.3;
   RL_LP_B4_L5_SG2 : ALIAS FOR ACNR_RP_SG_N4:6:O.4;
   RL_LP_B4_SG : ALIAS FOR ACNR_RP_SG_N4:5:O.2;
   RL_LP_ML_SG : ALIAS FOR ACNR_RP_SG_N4:1:O.0;
   SC_GP_BT_SG1 : ALIAS FOR ACNR_GP_SG_N2:3:O.0;
   SC_GP_BT_SG2 : ALIAS FOR ACNR_GP_SG_N2:3:O.1;
   SC_GP_GD_SG1 : ALIAS FOR ACNR_GP_SG_N2:3:O.2;
   SC_GP_GD_SG2 : ALIAS FOR ACNR_GP_SG_N2:3:O.3;
   SC_SP_LN_SG1 : ALIAS FOR ACNR_SP_SG_N3:2:O.2;
   SC_SP_LN_SG2 : ALIAS FOR ACNR_SP_SG_N3:2:O.3;
   Scenario : Scenario_Def[100] := ([1].Name := 'Source and Grid panels, all relays.', [1].Step[1].Output_Table.Data[1] := 16384, [1].Step[1].Configured_Step_Time := 5, [1].Step[2].Output_Table.Data[1] := 32768, [1].Step[2].Configured_Step_Time := 5, [1].Step[3].Output_Table.Data[1] := 4096, [1].Step[3].Configured_Step_Time := 5, [1].Step[4].Output_Table.Data[1] := 8192, [1].Step[4].Configured_Step_Time := 5, [1].Step[5].Output_Table.Data[1] := 1024, [1].Step[5].Configured_Step_Time := 5, [1].Step[6].Output_Table.Data[1] := 1024, [1].Step[6].Configured_Step_Time := 5, [1].Step[7].Output_Table.Data[1] := 256, [1].Step[7].Configured_Step_Time := 5, [1].Step[8].Output_Table.Data[1] := 512, [1].Step[8].Configured_Step_Time := 5, [1].Step[9].Output_Table.Data[1] := 64, [1].Step[9].Configured_Step_Time := 5, [1].Step[10].Output_Table.Data[1] := 128, [1].Step[10].Configured_Step_Time := 5, [1].Step[11].Output_Table.Data[1] := 16, [1].Step[11].Configured_Step_Time := 5, [1].Step[12].Output_Table.Data[1] := 32, [1].Step[12].Configured_Step_Time := 5, [1].Step[13].Output_Table.Data[1] := 4, [1].Step[13].Configured_Step_Time := 5, [1].Step[14].Output_Table.Data[1] := 8, [1].Step[14].Configured_Step_Time := 5, [1].Step[15].Output_Table.Data[1] := 1, [1].Step[15].Configured_Step_Time := 5, [1].Step[16].Output_Table.Data[1] := 2, [1].Step[16].Configured_Step_Time := 5, [1].Step[17].Output_Table.Data[0] := 64, [1].Step[17].Configured_Step_Time := 5, [1].Step[18].Output_Table.Data[0] := 128, [1].Step[18].Configured_Step_Time := 5, [1].Step[19].Output_Table.Data[0] := 16, [1].Step[19].Configured_Step_Time := 5, [1].Step[20].Output_Table.Data[0] := 32, [1].Step[20].Configured_Step_Time := 5, [1].Step[21].Output_Table.Data[0] := 1024, [1].Step[21].Configured_Step_Time := 5, [1].Step[22].Output_Table.Data[0] := 2048, [1].Step[22].Configured_Step_Time := 5, [1].Step[23].Output_Table.Data[0] := 256, [1].Step[23].Configured_Step_Time := 5, [1].Step[24].Output_Table.Data[0] := 512, [1].Step[24].Configured_Step_Time := 5, [1].Step[25].Output_Table.Data[0] := 16384, [1].Step[25].Configured_Step_Time := 5, [1].Step[26].Output_Table.Data[0] := 32768, [1].Step[26].Configured_Step_Time := 5, [1].Step[27].Output_Table.Data[0] := 4096, [1].Step[27].Configured_Step_Time := 5, [1].Step[28].Output_Table.Data[0] := 8192, [1].Step[28].Configured_Step_Time := 5, [1].Step[29].Output_Table.Data[0] := 262144, [1].Step[29].Configured_Step_Time := 5, [1].Step[30].Output_Table.Data[0] := 524288,
        [1].Step[30].Configured_Step_Time := 5, [1].Step[31].Output_Table.Data[0] := 65536, [1].Step[31].Configured_Step_Time := 5, [1].Step[32].Output_Table.Data[0] := 131072, [1].Step[32].Configured_Step_Time := 5, [1].Step[33].Output_Table.Data[0] := 1073741824, [1].Step[33].Configured_Step_Time := 5, [1].Step[34].Output_Table.Data[0] := -2147483648, [1].Step[34].Configured_Step_Time := 5, [1].Step[35].Output_Table.Data[0] := 268435456, [1].Step[35].Configured_Step_Time := 5, [1].Step[36].Output_Table.Data[0] := 536870912, [1].Step[36].Configured_Step_Time := 5, [1].Step[37].Output_Table.Data[0] := 67108864, [1].Step[37].Configured_Step_Time := 5, [1].Step[38].Output_Table.Data[0] := 134217728, [1].Step[38].Configured_Step_Time := 5, [1].Step[39].Output_Table.Data[0] := 16777216, [1].Step[39].Configured_Step_Time := 5, [1].Step[40].Output_Table.Data[0] := 33554432, [1].Step[40].Configured_Step_Time := 5, [1].Step[41].Output_Table.Data[0] := 1, [1].Step[41].Configured_Step_Time := 5, [1].Step[42].Output_Table.Data[0] := 2, [1].Step[42].Configured_Step_Time := 5, [1].Step[43].Output_Table.Data[0] := 4, [1].Step[43].Configured_Step_Time := 5, [1].Step[44].Output_Table.Data[0] := 8, [1].Step[44].Configured_Step_Time := 5, [1].Step[45].Output_Table.Data[2] := 1024, [1].Step[45].Configured_Step_Time := 35, [1].Step[46].Output_Table.Data[2] := 2048, [1].Step[46].Configured_Step_Time := 5, [1].Step[47].Output_Table.Data[2] := 256, [1].Step[47].Configured_Step_Time := 5, [1].Step[48].Output_Table.Data[2] := 512, [1].Step[48].Configured_Step_Time := 5, [1].Step[49].Output_Table.Data[2] := 64, [1].Step[49].Configured_Step_Time := 5, [1].Step[50].Output_Table.Data[2] := 128, [1].Step[50].Configured_Step_Time := 5, [1].Step[51].Output_Table.Data[2] := 16, [1].Step[51].Configured_Step_Time := 5, [1].Step[52].Output_Table.Data[2] := 32, [1].Step[52].Configured_Step_Time := 5, [1].Step[53].Output_Table.Data[2] := 4, [1].Step[53].Configured_Step_Time := 5, [1].Step[54].Output_Table.Data[2] := 8, [1].Step[54].Configured_Step_Time := 5, [1].Step[55].Output_Table.Data[2] := 1, [1].Step[55].Configured_Step_Time := 5, [1].Step[56].Output_Table.Data[2] := 2, [1].Step[56].Configured_Step_Time := 5, [2].Name := 'Load panels, load relays only.', [2].Step[1].Output_Table.Data[4] := 4, [2].Step[1].Configured_Step_Time := 5, [2].Step[2].Output_Table.Data[4] := 8, [2].Step[2].Configured_Step_Time := 5, [2].Step[3].Output_Table.Data[4] := 16, [2].Step[3].Configured_Step_Time := 5,
        [2].Step[4].Output_Table.Data[4] := 32, [2].Step[4].Configured_Step_Time := 5, [2].Step[5].Output_Table.Data[4] := 64, [2].Step[5].Configured_Step_Time := 5, [2].Step[6].Output_Table.Data[4] := 128, [2].Step[6].Configured_Step_Time := 5, [2].Step[7].Output_Table.Data[4] := 256, [2].Step[7].Configured_Step_Time := 5, [2].Step[8].Output_Table.Data[4] := 512, [2].Step[8].Configured_Step_Time := 5, [2].Step[9].Output_Table.Data[4] := 1024, [2].Step[9].Configured_Step_Time := 5, [2].Step[10].Output_Table.Data[4] := 2048, [2].Step[10].Configured_Step_Time := 5, [2].Step[11].Output_Table.Data[4] := 8192, [2].Step[11].Configured_Step_Time := 5, [2].Step[12].Output_Table.Data[4] := 16384, [2].Step[12].Configured_Step_Time := 5, [2].Step[13].Output_Table.Data[4] := 32768, [2].Step[13].Configured_Step_Time := 5, [2].Step[14].Output_Table.Data[4] := 65536, [2].Step[14].Configured_Step_Time := 5, [2].Step[15].Output_Table.Data[4] := 131072, [2].Step[15].Configured_Step_Time := 5, [2].Step[16].Output_Table.Data[4] := 262144, [2].Step[16].Configured_Step_Time := 5, [2].Step[17].Output_Table.Data[4] := 524288, [2].Step[17].Configured_Step_Time := 5, [2].Step[18].Output_Table.Data[4] := 1048576, [2].Step[18].Configured_Step_Time := 5, [2].Step[19].Output_Table.Data[4] := 2097152, [2].Step[19].Configured_Step_Time := 5, [2].Step[20].Output_Table.Data[4] := 4194304, [2].Step[20].Configured_Step_Time := 5, [2].Step[21].Output_Table.Data[4] := 16777216, [2].Step[21].Configured_Step_Time := 5, [2].Step[22].Output_Table.Data[4] := 33554432, [2].Step[22].Configured_Step_Time := 5, [2].Step[23].Output_Table.Data[4] := 67108864, [2].Step[23].Configured_Step_Time := 5, [2].Step[24].Output_Table.Data[4] := 134217728, [2].Step[24].Configured_Step_Time := 5, [2].Step[25].Output_Table.Data[4] := 268435456, [2].Step[25].Configured_Step_Time := 5, [2].Step[26].Output_Table.Data[4] := 536870912, [2].Step[26].Configured_Step_Time := 5, [2].Step[27].Output_Table.Data[4] := 1073741824, [2].Step[27].Configured_Step_Time := 5, [2].Step[28].Output_Table.Data[4] := -2147483648, [2].Step[28].Configured_Step_Time := 5, [2].Step[29].Output_Table.Data[5] := 1, [2].Step[29].Configured_Step_Time := 5, [2].Step[30].Output_Table.Data[5] := 2, [2].Step[30].Configured_Step_Time := 5, [2].Step[31].Output_Table.Data[5] := 8, [2].Step[31].Configured_Step_Time := 5, [2].Step[32].Output_Table.Data[5] := 16, [2].Step[32].Configured_Step_Time := 5, [2].Step[33].Output_Table.Data[5] := 32, [2].Step[33].Configured_Step_Time := 5,
        [2].Step[34].Output_Table.Data[5] := 64, [2].Step[34].Configured_Step_Time := 5, [2].Step[35].Output_Table.Data[5] := 128, [2].Step[35].Configured_Step_Time := 5, [2].Step[36].Output_Table.Data[5] := 256, [2].Step[36].Configured_Step_Time := 5, [2].Step[37].Output_Table.Data[5] := 512, [2].Step[37].Configured_Step_Time := 5, [2].Step[38].Output_Table.Data[5] := 1024, [2].Step[38].Configured_Step_Time := 5, [2].Step[39].Output_Table.Data[5] := 2048, [2].Step[39].Configured_Step_Time := 5, [2].Step[40].Output_Table.Data[5] := 4096, [2].Step[40].Configured_Step_Time := 5, [2].Step[41].Output_Table.Data[7] := 32, [2].Step[41].Configured_Step_Time := 35, [2].Step[42].Output_Table.Data[7] := 64, [2].Step[42].Configured_Step_Time := 5, [2].Step[43].Output_Table.Data[7] := 256, [2].Step[43].Configured_Step_Time := 5, [2].Step[44].Output_Table.Data[7] := 512, [2].Step[44].Configured_Step_Time := 5, [2].Step[45].Output_Table.Data[7] := 1024, [2].Step[45].Configured_Step_Time := 5, [2].Step[46].Output_Table.Data[7] := 2048, [2].Step[46].Configured_Step_Time := 5, [2].Step[47].Output_Table.Data[7] := 4096, [2].Step[47].Configured_Step_Time := 5, [2].Step[48].Output_Table.Data[7] := 8192, [2].Step[48].Configured_Step_Time := 5, [2].Step[49].Output_Table.Data[7] := 16384, [2].Step[49].Configured_Step_Time := 5, [2].Step[50].Output_Table.Data[7] := 32768, [2].Step[50].Configured_Step_Time := 5, [2].Step[51].Output_Table.Data[6] := 67108864, [2].Step[51].Configured_Step_Time := 5, [2].Step[52].Output_Table.Data[6] := 134217728, [2].Step[52].Configured_Step_Time := 5, [2].Step[53].Output_Table.Data[6] := 268435456, [2].Step[53].Configured_Step_Time := 5, [2].Step[54].Output_Table.Data[6] := 536870912, [2].Step[54].Configured_Step_Time := 5, [2].Step[55].Output_Table.Data[6] := 1073741824, [2].Step[55].Configured_Step_Time := 5, [2].Step[56].Output_Table.Data[6] := -2147483648, [2].Step[56].Configured_Step_Time := 5, [2].Step[57].Output_Table.Data[7] := 1, [2].Step[57].Configured_Step_Time := 5, [2].Step[58].Output_Table.Data[7] := 2, [2].Step[58].Configured_Step_Time := 5, [2].Step[59].Output_Table.Data[7] := 4, [2].Step[59].Configured_Step_Time := 5, [2].Step[60].Output_Table.Data[7] := 8, [2].Step[60].Configured_Step_Time := 5, [2].Step[61].Output_Table.Data[6] := 8192, [2].Step[61].Configured_Step_Time := 5, [2].Step[62].Output_Table.Data[6] := 16384, [2].Step[62].Configured_Step_Time := 5, [2].Step[63].Output_Table.Data[6] := 65536, [2].Step[63].Configured_Step_Time := 5,
        [2].Step[64].Output_Table.Data[6] := 131072, [2].Step[64].Configured_Step_Time := 5, [2].Step[65].Output_Table.Data[6] := 262144, [2].Step[65].Configured_Step_Time := 5, [2].Step[66].Output_Table.Data[6] := 524288, [2].Step[66].Configured_Step_Time := 5, [2].Step[67].Output_Table.Data[6] := 1048576, [2].Step[67].Configured_Step_Time := 5, [2].Step[68].Output_Table.Data[6] := 2097152, [2].Step[68].Configured_Step_Time := 5, [2].Step[69].Output_Table.Data[6] := 4194304, [2].Step[69].Configured_Step_Time := 5, [2].Step[70].Output_Table.Data[6] := 8388608, [2].Step[70].Configured_Step_Time := 5, [2].Step[71].Output_Table.Data[6] := 4, [2].Step[71].Configured_Step_Time := 5, [2].Step[72].Output_Table.Data[6] := 8, [2].Step[72].Configured_Step_Time := 5, [2].Step[73].Output_Table.Data[6] := 16, [2].Step[73].Configured_Step_Time := 5, [2].Step[74].Output_Table.Data[6] := 32, [2].Step[74].Configured_Step_Time := 5, [2].Step[75].Output_Table.Data[6] := 64, [2].Step[75].Configured_Step_Time := 5, [2].Step[76].Output_Table.Data[6] := 128, [2].Step[76].Configured_Step_Time := 5, [2].Step[77].Output_Table.Data[6] := 256, [2].Step[77].Configured_Step_Time := 5, [2].Step[78].Output_Table.Data[6] := 512, [2].Step[78].Configured_Step_Time := 5, [2].Step[79].Output_Table.Data[6] := 1024, [2].Step[79].Configured_Step_Time := 5, [2].Step[80].Output_Table.Data[6] := 2048, [2].Step[80].Configured_Step_Time := 5, [3].Name := 'Load panels, ground fault relays only.', [3].Step[1].Output_Table.Data[4] := 1, [3].Step[1].Configured_Step_Time := 5, [3].Step[2].Output_Table.Data[4] := 2, [3].Step[2].Configured_Step_Time := 5, [3].Step[3].Output_Table.Data[4] := 4096, [3].Step[3].Configured_Step_Time := 5, [3].Step[4].Output_Table.Data[4] := 8388608, [3].Step[4].Configured_Step_Time := 5, [3].Step[5].Output_Table.Data[5] := 4, [3].Step[5].Configured_Step_Time := 5, [3].Step[6].Output_Table.Data[6] := 16777216, [3].Step[6].Configured_Step_Time := 35, [3].Step[7].Output_Table.Data[7] := 16, [3].Step[7].Configured_Step_Time := 5, [3].Step[8].Output_Table.Data[6] := 33554432, [3].Step[8].Configured_Step_Time := 5, [3].Step[9].Output_Table.Data[6] := 1, [3].Step[9].Configured_Step_Time := 5, [3].Step[10].Output_Table.Data[6] := 4096, [3].Step[10].Configured_Step_Time := 5, [3].Step[11].Output_Table.Data[6] := 2, [3].Step[11].Configured_Step_Time := 5, [4].Name := 'Scenario 04', [5].Name := 'Scenario 05', [6].Name := 'Scenario 06',
        [7].Name := 'Scenario 07', [8].Name := 'Scenario 08', [9].Name := 'Scenario 09', [10].Name := 'Scenario 10', [11].Name := 'Scenario 11', [12].Name := 'Scenario 12', [13].Name := 'Scenario 13', [14].Name := 'Scenario 14', [15].Name := 'Scenario 15', [16].Name := 'Scenario 16', [17].Name := 'Scenario 17', [18].Name := 'Scenario 18', [19].Name := 'Scenario 19', [20].Name := 'Scenario 20', [21].Name := 'Scenario 21', [22].Name := 'Scenario 22', [23].Name := 'Scenario 23', [24].Name := 'Scenario 24', [25].Name := 'Scenario 25', [26].Name := 'Scenario 26', [27].Name := 'Scenario 27', [28].Name := 'Scenario 28', [29].Name := 'Scenario 29', [30].Name := 'Scenario 30', [31].Name := 'Scenario 31', [32].Name := 'Scenario 32', [33].Name := 'Scenario 33', [34].Name := 'Scenario 34', [35].Name := 'Scenario 35', [36].Name := 'Scenario 36', [37].Name := 'Scenario 37', [38].Name := 'Scenario 38', [39].Name := 'Scenario 39', [40].Name := 'Scenario 40', [41].Name := 'Scenario 41', [42].Name := 'Scenario 42', [43].Name := 'Scenario 43', [44].Name := 'Scenario 44', [45].Name := 'Scenario 45', [46].Name := 'Scenario 46', [47].Name := 'Scenario 47', [48].Name := 'Scenario 48', [49].Name := 'Scenario 49', [50].Name := 'Scenario 50', [51].Name := 'Scenario 51', [52].Name := 'Scenario 52', [53].Name := 'Scenario 53', [54].Name := 'Scenario 54', [55].Name := 'Scenario 55', [56].Name := 'Scenario 56', [57].Name := 'Scenario 57', [58].Name := 'Scenario 58', [59].Name := 'Scenario 59', [60].Name := 'Scenario 60', [61].Name := 'Scenario 61', [62].Name := 'Scenario 62', [63].Name := 'Scenario 63', [64].Name := 'Scenario 64', [65].Name := 'Scenario 65', [66].Name := 'Scenario 66',
        [67].Name := 'Scenario 67', [68].Name := 'Scenario 68', [69].Name := 'Scenario 69', [70].Name := 'Scenario 70', [71].Name := 'Scenario 71', [72].Name := 'Scenario 72', [73].Name := 'Scenario 73', [74].Name := 'Scenario 74', [75].Name := 'Scenario 75', [76].Name := 'Scenario 76', [77].Name := 'Scenario 77', [78].Name := 'Scenario 78', [79].Name := 'Scenario 79', [80].Name := 'Scenario 80', [81].Name := 'Scenario 81', [82].Name := 'Scenario 82', [83].Name := 'Scenario 83', [84].Name := 'Scenario 84', [85].Name := 'Scenario 85', [86].Name := 'Scenario 86', [87].Name := 'Scenario 87', [88].Name := 'Scenario 88', [89].Name := 'Scenario 89', [90].Name := 'Scenario 90', [91].Name := 'Scenario 91', [92].Name := 'Scenario 92', [93].Name := 'Scenario 93', [94].Name := 'Scenario 94', [95].Name := 'Scenario 95', [96].Name := 'Scenario 96', [97].Name := 'Scenario 97', [98].Name := 'Scenario 98', [99].Name := 'Scenario 99');
   Scenario_Mode : BOOL;
   SF_GP_BT_SG1 : ALIAS FOR ACNR_GP_SG_N2:2:O.4;
   SF_GP_BT_SG2 : ALIAS FOR ACNR_GP_SG_N2:2:O.5;
   SF_GP_GD_SG1 : ALIAS FOR ACNR_GP_SG_N2:2:O.6;
   SF_GP_GD_SG2 : ALIAS FOR ACNR_GP_SG_N2:2:O.7;
   SF_SP_LN_SG1 : ALIAS FOR ACNR_SP_SG_N3:2:O.0;
   SF_SP_LN_SG2 : ALIAS FOR ACNR_SP_SG_N3:2:O.1;
   TimeTblScenNmbr : DINT := 100;
   TimeTblStepNmbr : DINT := 100;
   WF_GP_BT_SG1 : ALIAS FOR ACNR_GP_SG_N2:1:O.4;
   WF_GP_BT_SG2 : ALIAS FOR ACNR_GP_SG_N2:1:O.5;
   WF_GP_GD_SG1 : ALIAS FOR ACNR_GP_SG_N2:1:O.6;
   WF_GP_GD_SG2 : ALIAS FOR ACNR_GP_SG_N2:1:O.7;
   WF_SP_LN_SG1 : ALIAS FOR ACNR_SP_SG_N3:1:O.4;
   WF_SP_LN_SG2 : ALIAS FOR ACNR_SP_SG_N3:1:O.5;
   WT_GP_BT_SG1 : ALIAS FOR ACNR_GP_SG_N2:2:O.0;
   WT_GP_BT_SG2 : ALIAS FOR ACNR_GP_SG_N2:2:O.1;
   WT_GP_GD_SG1 : ALIAS FOR ACNR_GP_SG_N2:2:O.2;
   WT_GP_GD_SG2 : ALIAS FOR ACNR_GP_SG_N2:2:O.3;
   WT_SP_LN_SG1 : ALIAS FOR ACNR_SP_SG_N3:1:O.6;
   WT_SP_LN_SG2 : ALIAS FOR ACNR_SP_SG_N3:1:O.7;
END_VAR

PROGRAM MainProgram   (* main routine MainRoutine *)
VAR
   ControlModePv : ControlModePv := (Cnx.Alternate_Control_Buffer.Data[1] := 1024, Comments[0] := 2047, Comments[1] := 53);
        .ONESHOT[0].0   // Alternate Control is Active One Shot
   DiscreteOutputsPv : DiscreteOutputsPv := (Comments[0] := 2047, Comments[1] := 53);
   EditScenarioPv : EditScenarioPv := (Comments[0] := 2047, Comments[1] := 61, Intrnl.Old_Scenario_Number := 3, Intrnl.Old_Scenario_Step := 3, Intrnl.Scenario_Name_Entered := 'Load panels, load relays only.', Intrnl.Scenario_Edit_Buffer.Output_Table.Data[4] := 4096, Intrnl.Scenario_Edit_Buffer.Configured_Step_Time := 5, Intrnl.Edit_Scenario_Number := 3, Intrnl.Edit_Step_Number := 3, Intrnl.Requested_Step_Time := 5, Intrnl.Step_Time_Diag_Timer.PRE := 5000, Intrnl.Step_Time_Diag_Timer.ACC := 5000, Intrnl.Edit_Prev_Step_Number := 2, OneShot[0] := 480);
        .EV.EXECUTEEVENTS.1   // Event 1 - Run Command
        .EV.EXECUTEEVENTS.2   // Event 2 - Pause Command
        .EV.EXECUTEEVENTS.3   // Event 3 - Resume Command
        .EV.EXECUTEEVENTS.4   // Event 4 - Stop Command
        .ST.1   // State 1 - Stopped
        .ST.2   // State 2 - Running
        .ST.3   // State 3 - Paused
        .ONESHOT[0].9   // Initial Configuration Screen is active One Shot
        .ONESHOT[0].1   // Gris Configuration Screen is active One Shot
        .ONESHOT[0].5   // Exit Grid Configuration Screen One Shot
        .ONESHOT[0].2   // Source Configuration Screen is active One Shot
        .ONESHOT[0].3   // Residential Configuration Screen is active One Shot
        .ONESHOT[0].4   // Industrial Configuration Screen is active One Shot
        .ONESHOT[0].6   // Exit Source Configuration Screen One Shot
        .ONESHOT[0].7   // Exit Residential Configuration Screen One Shot
        .ONESHOT[0].8   // Exit Industrial Configuration Screen One Shot
        .ONESHOT[0].10   // Go To Next Step Command One Shot
        .ONESHOT[0].11   // Copy Previous Step Grid One Shot
        .ONESHOT[0].12   // Copy Previous Step Source One Shot
        .ONESHOT[0].13   // Copy Previous Step Residential One Shot
        .ONESHOT[0].14   // Copy Previous Step Industrial One Shot
   ExecutePv : ExecutePv := (Comments[0] := 2099199, Comments[1] := 125, Intrnl.Current_Step_Number := 1, Intrnl.Current_Scenario_Number := 1, Intrnl.Scenario_Start_Number := 1, Intrnl.Scenario_Stop_Number := 2, Intrnl.Step_Start_Number := 1, Intrnl.Step_Stop_Number := 80, Intrnl.Time_Multiplier := 10, Intrnl.Total_Scenario_Time_Config := 740, Intrnl.Scenario_Time_Remaining_Config := 735, Intrnl.Total_Step_Time_Config := 5, Intrnl.Total_Scenario_Time_Actual := 7400, Intrnl.Scenario_Time_Remaining_Actual := 7350, Intrnl.Total_Step_Time_Actual := 50, Intrnl.Virtual_Start_Step := 101, Intrnl.Virtual_Stop_Step := 280, Intrnl.Virtual_Current_Step := 101, Intrnl.Virtual_Current_Step_Plus_1 := 102, Intrnl.Requested_Scenario_Start_Number := 1, Intrnl.Requested_Scenario_Stop_Number := 2, Intrnl.Requested_Step_Start_Number := 1, Intrnl.Requested_Step_Stop_Number := 80, Intrnl.Requested_Time_Multiplier := 10, Intrnl.Requested_Virtual_Start_Step := 101, Intrnl.Requested_Virtual_Stop_Step := 280, Intrnl.TM_Diag_Timer.PRE := 5000, Intrnl.TM_Diag_Timer.ACC := 5000, Intrnl.SAS_Diag_Timer.PRE := 5000, Intrnl.SAS_Diag_Timer.ACC := 5003, Intrnl.SBS_Diag_Timer.PRE := 5000, Intrnl.SBS_Diag_Timer.ACC := 5000, Intrnl.Start_Scenario_Diag_Timer.PRE := 5000, Intrnl.Start_Scenario_Diag_Timer.ACC := 5000, Intrnl.Stop_Scenario_Diag_Timer.PRE := 5000, Intrnl.Stop_Scenario_Diag_Timer.ACC := 5000, Intrnl.Start_Step_Diag_Timer.PRE := 5000, Intrnl.Start_Step_Diag_Timer.ACC := 5000, Intrnl.Stop_Step_Diag_Timer.PRE := 5000, Intrnl.Stop_Step_Diag_Timer.ACC := 5000, Intrnl.VirtualStepTime[101] := 5, Intrnl.VirtualStepTime[102] := 5, Intrnl.VirtualStepTime[103] := 5, Intrnl.VirtualStepTime[104] := 5, Intrnl.VirtualStepTime[105] := 5, Intrnl.VirtualStepTime[106] := 5, Intrnl.VirtualStepTime[107] := 5, Intrnl.VirtualStepTime[108] := 5, Intrnl.VirtualStepTime[109] := 5, Intrnl.VirtualStepTime[110] := 5, Intrnl.VirtualStepTime[111] := 5, Intrnl.VirtualStepTime[112] := 5, Intrnl.VirtualStepTime[113] := 5, Intrnl.VirtualStepTime[114] := 5, Intrnl.VirtualStepTime[115] := 5, Intrnl.VirtualStepTime[116] := 5, Intrnl.VirtualStepTime[117] := 5, Intrnl.VirtualStepTime[118] := 5, Intrnl.VirtualStepTime[119] := 5, Intrnl.VirtualStepTime[120] := 5,
        Intrnl.VirtualStepTime[121] := 5, Intrnl.VirtualStepTime[122] := 5, Intrnl.VirtualStepTime[123] := 5, Intrnl.VirtualStepTime[124] := 5, Intrnl.VirtualStepTime[125] := 5, Intrnl.VirtualStepTime[126] := 5, Intrnl.VirtualStepTime[127] := 5, Intrnl.VirtualStepTime[128] := 5, Intrnl.VirtualStepTime[129] := 5, Intrnl.VirtualStepTime[130] := 5, Intrnl.VirtualStepTime[131] := 5, Intrnl.VirtualStepTime[132] := 5, Intrnl.VirtualStepTime[133] := 5, Intrnl.VirtualStepTime[134] := 5, Intrnl.VirtualStepTime[135] := 5, Intrnl.VirtualStepTime[136] := 5, Intrnl.VirtualStepTime[137] := 5, Intrnl.VirtualStepTime[138] := 5, Intrnl.VirtualStepTime[139] := 5, Intrnl.VirtualStepTime[140] := 5, Intrnl.VirtualStepTime[141] := 5, Intrnl.VirtualStepTime[142] := 5, Intrnl.VirtualStepTime[143] := 5, Intrnl.VirtualStepTime[144] := 5, Intrnl.VirtualStepTime[145] := 35, Intrnl.VirtualStepTime[146] := 5, Intrnl.VirtualStepTime[147] := 5, Intrnl.VirtualStepTime[148] := 5, Intrnl.VirtualStepTime[149] := 5, Intrnl.VirtualStepTime[150] := 5, Intrnl.VirtualStepTime[151] := 5, Intrnl.VirtualStepTime[152] := 5, Intrnl.VirtualStepTime[153] := 5, Intrnl.VirtualStepTime[154] := 5, Intrnl.VirtualStepTime[155] := 5, Intrnl.VirtualStepTime[156] := 5, Intrnl.VirtualStepTime[201] := 5, Intrnl.VirtualStepTime[202] := 5, Intrnl.VirtualStepTime[203] := 5, Intrnl.VirtualStepTime[204] := 5, Intrnl.VirtualStepTime[205] := 5, Intrnl.VirtualStepTime[206] := 5, Intrnl.VirtualStepTime[207] := 5, Intrnl.VirtualStepTime[208] := 5, Intrnl.VirtualStepTime[209] := 5, Intrnl.VirtualStepTime[210] := 5, Intrnl.VirtualStepTime[211] := 5, Intrnl.VirtualStepTime[212] := 5, Intrnl.VirtualStepTime[213] := 5, Intrnl.VirtualStepTime[214] := 5, Intrnl.VirtualStepTime[215] := 5, Intrnl.VirtualStepTime[216] := 5, Intrnl.VirtualStepTime[217] := 5, Intrnl.VirtualStepTime[218] := 5, Intrnl.VirtualStepTime[219] := 5, Intrnl.VirtualStepTime[220] := 5, Intrnl.VirtualStepTime[221] := 5, Intrnl.VirtualStepTime[222] := 5, Intrnl.VirtualStepTime[223] := 5, Intrnl.VirtualStepTime[224] := 5,
        Intrnl.VirtualStepTime[225] := 5, Intrnl.VirtualStepTime[226] := 5, Intrnl.VirtualStepTime[227] := 5, Intrnl.VirtualStepTime[228] := 5, Intrnl.VirtualStepTime[229] := 5, Intrnl.VirtualStepTime[230] := 5, Intrnl.VirtualStepTime[231] := 5, Intrnl.VirtualStepTime[232] := 5, Intrnl.VirtualStepTime[233] := 5, Intrnl.VirtualStepTime[234] := 5, Intrnl.VirtualStepTime[235] := 5, Intrnl.VirtualStepTime[236] := 5, Intrnl.VirtualStepTime[237] := 5, Intrnl.VirtualStepTime[238] := 5, Intrnl.VirtualStepTime[239] := 5, Intrnl.VirtualStepTime[240] := 5, Intrnl.VirtualStepTime[241] := 35, Intrnl.VirtualStepTime[242] := 5, Intrnl.VirtualStepTime[243] := 5, Intrnl.VirtualStepTime[244] := 5, Intrnl.VirtualStepTime[245] := 5, Intrnl.VirtualStepTime[246] := 5, Intrnl.VirtualStepTime[247] := 5, Intrnl.VirtualStepTime[248] := 5, Intrnl.VirtualStepTime[249] := 5, Intrnl.VirtualStepTime[250] := 5, Intrnl.VirtualStepTime[251] := 5, Intrnl.VirtualStepTime[252] := 5, Intrnl.VirtualStepTime[253] := 5, Intrnl.VirtualStepTime[254] := 5, Intrnl.VirtualStepTime[255] := 5, Intrnl.VirtualStepTime[256] := 5, Intrnl.VirtualStepTime[257] := 5, Intrnl.VirtualStepTime[258] := 5, Intrnl.VirtualStepTime[259] := 5, Intrnl.VirtualStepTime[260] := 5, Intrnl.VirtualStepTime[261] := 5, Intrnl.VirtualStepTime[262] := 5, Intrnl.VirtualStepTime[263] := 5, Intrnl.VirtualStepTime[264] := 5, Intrnl.VirtualStepTime[265] := 5, Intrnl.VirtualStepTime[266] := 5, Intrnl.VirtualStepTime[267] := 5, Intrnl.VirtualStepTime[268] := 5, Intrnl.VirtualStepTime[269] := 5, Intrnl.VirtualStepTime[270] := 5, Intrnl.VirtualStepTime[271] := 5, Intrnl.VirtualStepTime[272] := 5, Intrnl.VirtualStepTime[273] := 5, Intrnl.VirtualStepTime[274] := 5, Intrnl.VirtualStepTime[275] := 5, Intrnl.VirtualStepTime[276] := 5, Intrnl.VirtualStepTime[277] := 5, Intrnl.VirtualStepTime[278] := 5, Intrnl.VirtualStepTime[279] := 5, Intrnl.VirtualStepTime[280] := 5, Intrnl.VirtualStepTime[301] := 5, Intrnl.VirtualStepTime[302] := 5, Intrnl.VirtualStepTime[303] := 5, Intrnl.VirtualStepTime[304] := 5,
        Intrnl.VirtualStepTime[305] := 5, Intrnl.VirtualStepTime[306] := 35, Intrnl.VirtualStepTime[307] := 5, Intrnl.VirtualStepTime[308] := 5, Intrnl.VirtualStepTime[309] := 5, Intrnl.VirtualStepTime[310] := 5, Intrnl.VirtualStepTime[311] := 5, Intrnl.BuildTableScanCounter := 24, OneShot[0] := 5, St := 2);
        .EV.EXECUTEEVENTS.1   // Event 1 - Run Command
        .EV.EXECUTEEVENTS.2   // Event 2 - Pause Command
        .EV.EXECUTEEVENTS.3   // Event 3 - Resume Command
        .EV.EXECUTEEVENTS.4   // Event 4 - Stop Command
        .ST.1   // State 1 - Stopped
        .ST.2   // State 2 - Running
        .ST.3   // State 3 - Paused
        .ONESHOT[0].1   // Skip Command One Shot
        .ONESHOT[0].0   // Program is Stopped One Shot
   HMIPv : HMIPv := (Comments[0] := 4095, Comments[1] := 1);
END_VAR
